Fanuc KAREL source: ka00055.KL

-- PROVISIONAL review KL for V1013-1; original PC SHA256 aee8d1a46f97cc60a59893521e5268f8efbcc49be73f6902403d1a300ad0fd7a
-- Incomplete behavior may be omitted. Consult companion uncertainty JSON. Do not deploy.
PROGRAM KA00055
%NOLOCKGROUP
-- UNRESOLVED_DECL SRC type=000101
-- UNRESOLVED_DECL DST type=000106
BEGIN
  -- UNRESOLVED_PC offsets 5-25; opcodes 49,7E,4A
  -- UNRESOLVED_PC offsets 30-34; opcodes 7F
END KA00055
